DATA_BLOCK "dbArchiveEquipBoiler"
{ S7_Optimized_Access := 'TRUE' }
VERSION : 0.8
"fbArchiveEquipBoiler"

BEGIN

END_DATA_BLOCK

